FUNCTION_BLOCK RT_E_CYCLE (* Delayed propagation of an event-Cancellable *)
  (* Standard: 61499-1; Classification: Event processing *)
  (* Version 0.0, 2008-07-10, 4DIAC-IDE, 4DIAC-Consortium *)
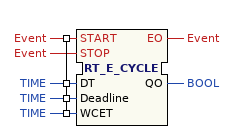
  EVENT_INPUT
    START WITH DT, Deadline, WCET; (* Begin Delay *)
    STOP; (* Cancel Delay *)
  END_EVENT
  EVENT_OUTPUT
    EO; (* Delayed Event *)
  END_EVENT
  VAR_INPUT
    DT : TIME; (* Delay Time *)
    Deadline : TIME;
    WCET : TIME;
  END_VAR
  VAR_OUTPUT
    QO : BOOL;
  END_VAR
END_FUNCTION_BLOCK
